FUNCTION_BLOCK FB_Enable_Motion
VAR_INPUT
	bAutoSwitch								: BOOL;
	bStartButton							: BOOL;
	
	eStatus									: BOOL;
	
	bManualSwitch							: BOOL;
	
	bPrimaryActive							: BOOL;
	bSecondaryActive						: BOOL;
	
END_VAR
VAR_OUTPUT
	bAutoEnable 							: BOOL;
	bManualEnable 							: BOOL; 
	bAutoEnable_SC 							: BOOL; 
	bManualEnable_SC					    : BOOL; 
END_VAR
VAR
END_VAR

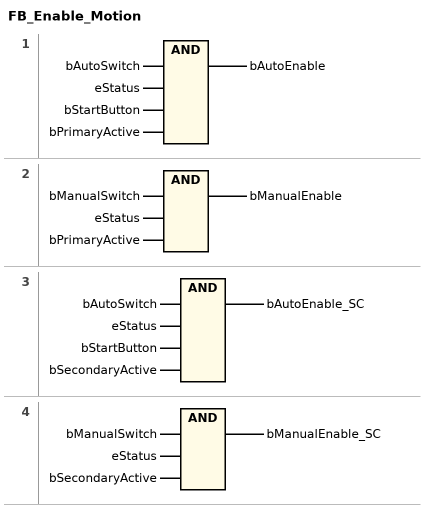
// NETWORK 1
bAutoEnable := bAutoSwitch AND eStatus AND bStartButton AND bPrimaryActive;

// NETWORK 2
bManualEnable := bManualSwitch AND eStatus AND bPrimaryActive;

// NETWORK 3
bAutoEnable_SC := bAutoSwitch AND eStatus AND bStartButton AND bSecondaryActive;

// NETWORK 4
bManualEnable_SC := bManualSwitch AND eStatus AND bSecondaryActive;

END_FUNCTION_BLOCK

(* stored: Version 1.1.0.1
   POU FB_Enable_Motion: Id {a65630a7-98e0-47b6-bc78-d4e9bb9c0bb6}, SpecialFunc None *)
